DATA_BLOCK "InstEM00_00_Main"   // DB31640
TITLE = instEM00_00_Main
AUTHOR : tech.team.motioncontrol@siemens.com
FAMILY : CPG
VERSION : 1.0
// Support: tech.team.motioncontrol@siemens.com
// Fax: +49 (0) 9131/98-1297
// stored: AutoNumber true, DBAccessibleFromOPCUA true, DBAccessibleFromWebserver true, InstanceOfName EM00_00_Main, InstanceOfType FB
"EM00_00_Main"
BEGIN
   // instEventControl.instEventMgr_Warning : instance FB - Event Manager - Warning Events
END_DATA_BLOCK

DATA_BLOCK "InstEM01_00_Main"   // DB31660
TITLE = InstEM01_00_Main
AUTHOR : tech.team.motioncontrol@siemens.com
FAMILY : CPG
VERSION : 1.0
// Support: tech.team.motioncontrol@siemens.com
// Fax: +49 (0) 9131/98-1297
// stored: AutoNumber true, DBAccessibleFromOPCUA true, DBAccessibleFromWebserver true, InstanceOfName EM01_00_Main, InstanceOfType FB
"EM01_00_Main"
BEGIN
END_DATA_BLOCK

DATA_BLOCK "InstEM02_00_Main"   // DB31680
TITLE = InstEM02_00_Main
AUTHOR : tech.team.motioncontrol@siemens.com
FAMILY : CPG
VERSION : 1.0
// Support: tech.team.motioncontrol@siemens.com
// Fax: +49 (0) 9131/98-1297
// stored: AutoNumber true, DBAccessibleFromOPCUA true, DBAccessibleFromWebserver true, InstanceOfName EM02_00_Main, InstanceOfType FB
"EM02_00_Main"
BEGIN
END_DATA_BLOCK

DATA_BLOCK "InstUN_00_Main"   // DB31620
TITLE = instUN00_00_Main
AUTHOR : tech.team.motioncontrol@siemens.com
FAMILY : CPG
VERSION : 1.0
// Support: tech.team.motioncontrol@siemens.com
// Fax: +49 (0) 9131/98-1297
// stored: AutoNumber true, DBAccessibleFromOPCUA true, DBAccessibleFromWebserver true, InstanceOfName UN_00_Main, InstanceOfType FB
"UN_00_Main"
BEGIN
END_DATA_BLOCK
